(* CODESYS project SharedMemCom.ecp

Project tree, tasks and I/O mapping:
  Controller : 750-8212 PFC200 2ETH RS, WAGO, order no. 0750-8212, version 5.14.3.11
    application Application
      libraries: ; WagoAppMem, 1.6.2.0 (WAGO)
      task MySHMTask (cyclic, interval 50 ms, priority 15) calls WagoShmApp
      program WagoShmApp [ST]
      data type MyOutputProcessImage
      data type MyInputProcessImage
      function block FbShm [ST]: pData
    Kbus : Kbus, WAGO, version 1.4.0.2
        unmapped channels: K-BUS diagnostics
    MODBUS
      MODBUS : MODBUS, WAGO, order no. n/a, version 1.1.1.15
    Common.PCI
    Serial
      COM1 : COM1, WAGO, version 0.0.0.19
*)

// Controller/Application/MyOutputProcessImage
{attribute 'pack_mode' := '0'}
TYPE MyOutputProcessImage :
STRUCT
	
i1 : INT;


END_STRUCT
END_TYPE

// Controller/Application/MyInputProcessImage
{attribute 'pack_mode' := '0'}
TYPE MyInputProcessImage :
STRUCT
	
i1 : INT;


END_STRUCT
END_TYPE

// Controller/Application/WagoShmApp
PROGRAM WagoShmApp
VAR

FbShmForWriting  :	FbShm;
FbShmForReading  :	FbShm;
MyInputProcessImage : MyInputProcessImage;
MyOutputProcessImage : MyOutputProcessImage;
pMyInputProcessImage: POINTER TO MyInputProcessImage;
pMyOutputProcessImage: POINTER TO MyOutputProcessImage;
iCnt : INT;
iCnt2 : INT;
eResult: eResultCode;
eResult2: eResultCode;
xRequiresSystemMemory : BOOL := FALSE;
xAssumeExisting : BOOL;
xShmReadOpen : BOOL;
xShmWriteOpen : BOOL;
iMyData : INT := 1;
xCloseResult: eResultCode;
xClose: BOOL;
xOpen : BOOL;
END_VAR



IF xOpen THEN
	eResult := FbShmForWriting.OpenByName(sName:= '_CODESYS_SharedMemoryTest_Write', udiSize:= SIZEOF(MyInputProcessImage), xRequiresSystemMemory:= xRequiresSystemMemory, xAssumeExisting:= xAssumeExisting);
	eResult2 := FbShmForReading.OpenByName(sName:= '_CODESYS_SharedMemoryTest_Read', udiSize:= SIZEOF(MyOutputProcessImage), xRequiresSystemMemory:= xRequiresSystemMemory, xAssumeExisting:= xAssumeExisting);
	IF FbShmForWriting.IsOpen AND FbShmForReading.IsOpen THEN
		xOpen := FALSE;
		xShmReadOpen := TRUE;
		xShmWriteOpen := TRUE;
	ELSE
		xShmReadOpen := FALSE;
		xShmWriteOpen := FALSE;	
	END_IF
END_IF

IF xShmWriteOpen AND NOT xClose THEN
	pMyInputProcessImage := FbShmForWriting.pData;
	pMyInputProcessImage^.i1 := iMyData;
END_IF

IF xShmReadOpen AND NOT xClose THEN
	pMyOutputProcessImage := FbShmForReading.pData;
	pMyOutputProcessImage^.i1;
END_IF

IF xClose THEN
	xCloseResult := FbShmForWriting.Close();
	xCloseResult := FbShmForReading.Close();
	xShmReadOpen := FALSE;
	xShmWriteOpen := FALSE;	

END_IF

END_PROGRAM

// Controller/Application/FbShm
FUNCTION_BLOCK FbShm EXTENDS WagoAppMem.FbSharedMemory_Base
VAR_INPUT
END_VAR
VAR_OUTPUT
END_VAR
VAR
END_VAR

super^();

PROPERTY pData : pointer to MyInputProcessImage
GET
pData := GetDataPointer();
END_GET
SET
END_SET
END_PROPERTY

END_FUNCTION_BLOCK
